// TIA Portal V16 export
// export: Created 2021-08-06T10:12:21.2195005Z, ExportSetting WithDefaults, DisplayName Totally Integrated Automation Portal, DisplayVersion V16, DisplayName TIA Portal Version Control Interface, DisplayVersion V16, DisplayName TIA Portal Openness, DisplayVersion V16, DisplayName SINAMICS Startdrive Advanced, DisplayVersion V16 Update 1, DisplayName SINAMICS Startdrive G130, G150, S120, S150, SINAMICS MV, S210, DisplayVersion V16 Update 1, DisplayName SINAMICS Startdrive G110M, G120, G120C, G120D, G120P, DisplayVersion V16 Update 1, DisplayName STEP 7 Professional, DisplayVersion V16, DisplayName STEP 7 Safety, DisplayVersion V16, DisplayName WinCC Advanced, DisplayVersion V16
FUNCTION_BLOCK "@FB Template Lvl1"   // FB13, LAD
{ S7_Optimized_Access := 'TRUE' }
VERSION : 0.1
// stored: AutoNumber true, IsIECCheckEnabled false, IsRetainMemResEnabled false, MemoryReserve 100, SetENOAutomatically false, UDAEnableTagReadback false
   VAR_INPUT
      iDummyInput { ExternalAccessible := 'False'; ExternalVisible := 'False'; ExternalWritable := 'False'} : Bool;   // Input dummy
   END_VAR
   VAR_OUTPUT
      oDummyOutput { ExternalAccessible := 'False'; ExternalVisible := 'False'; ExternalWritable := 'False'} : Bool;   // Output dummy
   END_VAR
   VAR
      Data { S7_SetPoint := 'True'} : "UDT Data Template lvl1";   // Standard data
   END_VAR
   VAR RETAIN
      RData { S7_SetPoint := 'True'} : "UDT RData Template lvl1";   // Retain Data (saved after PLC restart)
   END_VAR
   VAR
      sChangeLanguage { ExternalAccessible := 'False'; ExternalVisible := 'False'; ExternalWritable := 'False'} : Bool;   // Check for language change
      PositiveEdge { ExternalAccessible := 'False'; ExternalVisible := 'False'; ExternalWritable := 'False'; S7_SetPoint := 'True'} : Array[1..3] of R_TRIG;   // Positive edge alarms
      NegativeEdge { ExternalAccessible := 'False'; ExternalVisible := 'False'; ExternalWritable := 'False'; S7_SetPoint := 'True'} : Array[1..3] of F_TRIG;   // Negative edge alarms
      AlarmDummy { ExternalAccessible := 'False'; ExternalVisible := 'False'; ExternalWritable := 'False'; S7_SetPoint := 'True'} : Program_Alarm;   // Alarm: Dummy alarm
   END_VAR
   VAR_TEMP
      dummyCondition : Bool;   // Temp dummy condition
   END_VAR
   VAR CONSTANT
      cAlarmDummy : Int := 1;   // Array index of alarm
      cWarningCommissioningModeHMI : Int := 2;   // Array index of alarm
      cMessageOutOfService : Int := 3;   // Array index of alarm
   END_VAR
BEGIN

REGION Network 1 (SCL): Alarms
   //*************************************************************************************************//
   //*                                                                                               *//
   //*                               Alarms and warnings handling                                    *//
   //*                                                                                               *//
   //*  Reset all internal alarms and warnings                                                       *//
   //*  Set the specific module alarms and warnings                                                  *//
   //*  If there is an alarm or warning set the general alarm or warning bit                         *//
   //*                                                                                               *//
   //*************************************************************************************************//   

   // Reset all warning type alarms here
   #Data.AlarmsModule.WarningCommissioningModeHMI := False;
   #Data.Status.Warning := False;

   // Reset all message type alarms here
   #Data.AlarmsModule.MessageOutOfService := False;

   // SET DUMMY ALARM
   // Alarm: Dummy alarm
   IF #dummyCondition AND NOT #Data.AlarmsDisable.AlarmModuleAlarm THEN
       // MODIFY CONDITIONS AND ALARM ACCORDINGLY
       #Data.AlarmsModule.AlarmModuleAlarm := True;
       #Data.Status.Alarm := true;
   END_IF;

   // Warning: Module is set to commissioning mode from HMI panel
   IF #Data.CmdHMI.CommissioningMode THEN
       #Data.AlarmsModule.WarningCommissioningModeHMI := True;
       #Data.Status.Warning := True;
   END_IF;

   // SET OUT OF SERVICE ALARM
   // Message: Module is out of service (generates no alarms anymore)
   IF #RData.Settings.OutOfService THEN
       // RESET ALL ALARMS, WARNINGS AND MESSAGES HERE
       #Data.AlarmsModule.MessageOutOfService := NOT #Data.AlarmsDisable.MessageOutOfService;
       #Data.AlarmsModule.WarningCommissioningModeHMI := False;
       #Data.Status.Alarm := False;
       #Data.Status.Warning := False;
   END_IF;
END_REGION

REGION Network 2
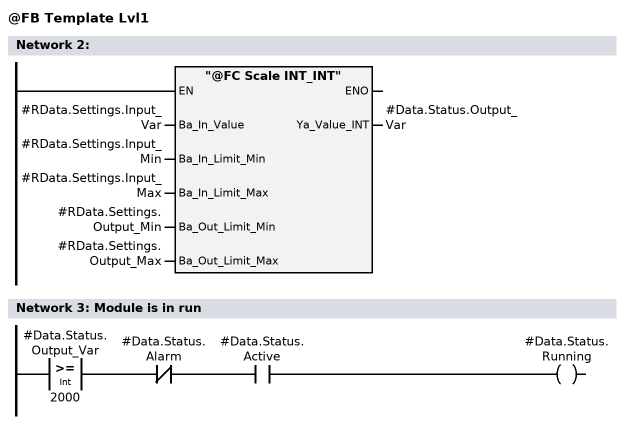
   RUNG wire#powerrail
      "@FC Scale INT_INT"(Ba_In_Value := #RData.Settings.Input_Var, Ba_In_Limit_Min := #RData.Settings.Input_Min, Ba_In_Limit_Max := #RData.Settings.Input_Max, Ba_Out_Limit_Min := #RData.Settings.Output_Min, Ba_Out_Limit_Max := #RData.Settings.Output_Max, Ya_Value_INT => #Data.Status.Output_Var)
   END_RUNG
   // the same network as SCL:
   "@FC Scale INT_INT"(Ba_In_Value := #RData.Settings.Input_Var,
                       Ba_In_Limit_Min := #RData.Settings.Input_Min,
                       Ba_In_Limit_Max := #RData.Settings.Input_Max,
                       Ba_Out_Limit_Min := #RData.Settings.Output_Min,
                       Ba_Out_Limit_Max := #RData.Settings.Output_Max,
                       Ya_Value_INT => #Data.Status.Output_Var);
END_REGION

REGION Network 3: Module is in run
   RUNG wire#powerrail
      { S7_Templates := "SrcType := Int" } GE_Contact(in1 := #Data.Status.Output_Var, in2 := 2000)
      I_Contact( #Data.Status.Alarm )
      Contact( #Data.Status.Active )
      Coil( #Data.Status.Running )
   END_RUNG
   // the same network as SCL:
   #Data.Status.Running := (#Data.Status.Output_Var >= 2000) AND NOT #Data.Status.Alarm AND #Data.Status.Active;
END_REGION

REGION Network 4 (SCL): Status
   //*************************************************************************************************//
   //*                                                                                               *//
   //*                                       Status handling                                         *//
   //*                                                                                               *//
   //*  Copy the tag name and the tag description                                                    *//
   //*  Copy the standard statuses from the upper level module                                       *//
   //*  Set/reset the HMI command buttons                                                            *//
   //*  Activate the module (Case statement for different modes)                                     *//              
   //*                                                                                               *//
   //*************************************************************************************************//     

   // Reset Output
   #Data.Status.Active := false;

   // Set Status Out of service
   #Data.Status.OutOfService := #RData.Settings.OutOfService;

   // Set Status Mode
   // Override Mode if commissioning bit in HMI is set
END_REGION
END_FUNCTION_BLOCK
